# B&R Automation Studio project Finale
Automation Studio 4.7.2.98

## Configuration Config1

### Hardware
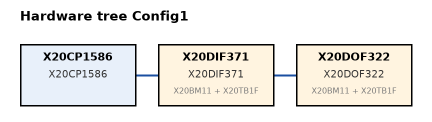
```
X20BM11a : X20BM11 v1.0.0.1  [X2X1 -> X20CP1586.IF6]
X20BM11b : X20BM11 v1.0.0.1  [X2X1 -> X20BM11a.X2X2]
X20CP1586 : X20CP1586 v1.8.0.0
  Connector IF2:
    ActivateDevice = 1
    Mode = Manual
    InternetAddress = 192.168.10.10
  Connector IF3:
    EplNatSubnet = 255.255.255.0
X20DIF371 : X20DIF371 v1.1.0.0  [SS1 -> X20TB1F1.SS; SL -> X20BM11a.SL1]
X20DOF322 : X20DOF322 v1.3.0.0  [SS1 -> X20TB1F2.SS; SL -> X20BM11b.SL1]
X20TB1F1 : X20TB1F v1.0.0.0
X20TB1F2 : X20TB1F v1.0.0.0
```

## Logical view

### Variables.var
```iecst
VAR
	controlPos0 : BOOL;
	controlPos1 : BOOL;
	controlPos2 : BOOL;
	rotaryMotor : BOOL;
	linearMotor : BOOL;
	gripper : BOOL;
	isSliderStateBit : BOOL;
	iRotaryMotionComplete : BOOL;
	slider : BOOL;
	iLinearMotionComplete : BOOL;
	prevFlag : USINT;
	flag : USINT;
	waitingFlag : BOOL;
	test : BOOL;
	destinationX : USINT;
	destinationY : USINT;
	sourceY : USINT;
	sourceX : USINT;
END_VAR
```
